// TIA Portal V21 export
FUNCTION "Motore_PompaMono" : Void   // FC133, LAD
{ S7_Optimized_Access := 'TRUE' }
// stored: SetENOAutomatically false
   VAR_TEMP
      AutoPos : Bool;
      AutoNeg : Bool;
   END_VAR
BEGIN

REGION Network 1: Comando positivo in automatico
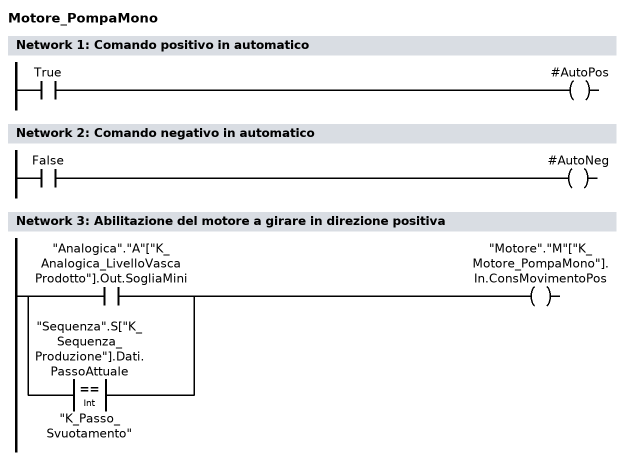
   RUNG wire#powerrail
      Contact( True )
      Coil( #AutoPos )
   END_RUNG
   // the same network as SCL:
   #AutoPos := True;
END_REGION

REGION Network 2: Comando negativo in automatico
   RUNG wire#powerrail
      Contact( False )
      Coil( #AutoNeg )
   END_RUNG
   // the same network as SCL:
   #AutoNeg := False;
END_REGION

REGION Network 3: Abilitazione del motore a girare in direzione positiva
   RUNG wire#powerrail
      Contact( "Analogica"."A"["K_Analogica_LivelloVascaProdotto"].Out.SogliaMini )
      wire#w1
      Coil( "Motore"."M"["K_Motore_PompaMono"].In.ConsMovimentoPos )
   END_RUNG
   RUNG wire#powerrail
      { S7_Templates := "SrcType := Int" } EQ_Contact(in1 := "Sequenza".S["K_Sequenza_Produzione"].Dati.PassoAttuale, in2 := "K_Passo_Svuotamento")
   END_RUNG wire#w1
   // the same network as SCL:
   "Motore"."M"["K_Motore_PompaMono"].In.ConsMovimentoPos := "Analogica"."A"["K_Analogica_LivelloVascaProdotto"].Out.SogliaMini OR ("Sequenza".S["K_Sequenza_Produzione"].Dati.PassoAttuale = "K_Passo_Svuotamento");
END_REGION

REGION Network 4 (SCL)
   REGION PompaMono
       REGION Ingressi
           "Motore".M[K_Motore_PompaMono].In.FbDigitali.FaultInverter := NOT "PompaMono_Ready";
           "Motore".M[K_Motore_PompaMono].In.FbDigitali.FeedbackMarcia := "PompaMono_Marcia";
           "Motore".M[K_Motore_PompaMono].In.ConsMovimentoPos := "Analogica".A[K_Analogica_LivelloVascaProdotto].Out.SogliaMini;
           //"Motore".M["K_Motore_PompaMono"].In.CmdPosRich := #AutoPos;
           //"Motore".M["K_Motore_PompaMono"].In.CmdNegRich := #AutoNeg;
           "Motore".M[K_Motore_PompaMono].Prm.Generali.K_Analogica := "K_Analogica_PortataIngressoProdotto";
       END_REGION ;
       REGION Gestione
           "GestMotore"(K_Motore := "K_Motore_PompaMono",
                        K_TipoMotore := "K_TipoMotore_InverterKEB",
                        K_Zona := "K_Zona_Sterilizzatore");

           "GestMotore_Servoventola"(K_Motore:="K_Motore_PompaMono",
                                     TermicoScattato:=NOT "PompaMono_Servoventola_TermicoOk",
                                     ComandoMarcia=>"PompaMono_ComandoServoventola");

       END_REGION ;
       REGION Uscite
           "PompaMono_ComandoMarcia" := "Motore".M[K_Motore_PompaMono].Out.CmdPosMotore;
           "PompaMono_Velocità" := DINT_TO_WORD("Motore".M[K_Motore_PompaMono].Out.Paw);
       END_REGION ;
   END_REGION ;
END_REGION
END_FUNCTION
